// SIMATIC S7-200 project (STEP 7-Micro/WIN), CPU 216 REL 01.02

SYMBOL_TABLE USR1
Always_On        SM0.0    // This bit is always on.
First_Scan_On    SM0.1    // This bit is on for the first scan cycle only.
Clock_1s         SM0.5    // Clock pulse that is on for 0.5 s, off for 0.5 s, for a duty cycle time of 1 s.
Down_Bit         M0.0     // This "count down" memory bit determines the counting direction.
END_SYMBOL_TABLE

ORGANIZATION_BLOCK MAIN:OB1
TITLE= Tip002B
//  题目： 处理输入/输出中断
// ***概述***
// 本程序适用于SIMATIC S7-212和S7-214的计数器，可以从0计到255，这要取决于输入I0.0
// 的状态。如果将输入I0.0置为1，则程序减计数；如果将输入I0.0置为0，则程序加计数
// 如果输入I0.0的状态改变，则将立即激活输入/输出中断程序，中断程序0或1分别将存储器位M0.0
// 置成1或0。
// ***程序和注释***
// 本程序是一个输入/输出中断程序的范例，计数器从0计到255。如果输入I0.0
// 为0，则程序加计数，如果输入I0.0为1，则程序减计数。
// 本程序包括以下三个程序：
// Main  （主程序）            初始化和计数
// INT0   （中断程序0）        输入I0.0为1时，减计数。
// INT1   （中断程序1）        输入I0.0为0时，加计数。
// 本程序长度为32个字。
// 标题：事件中断
// 
BEGIN
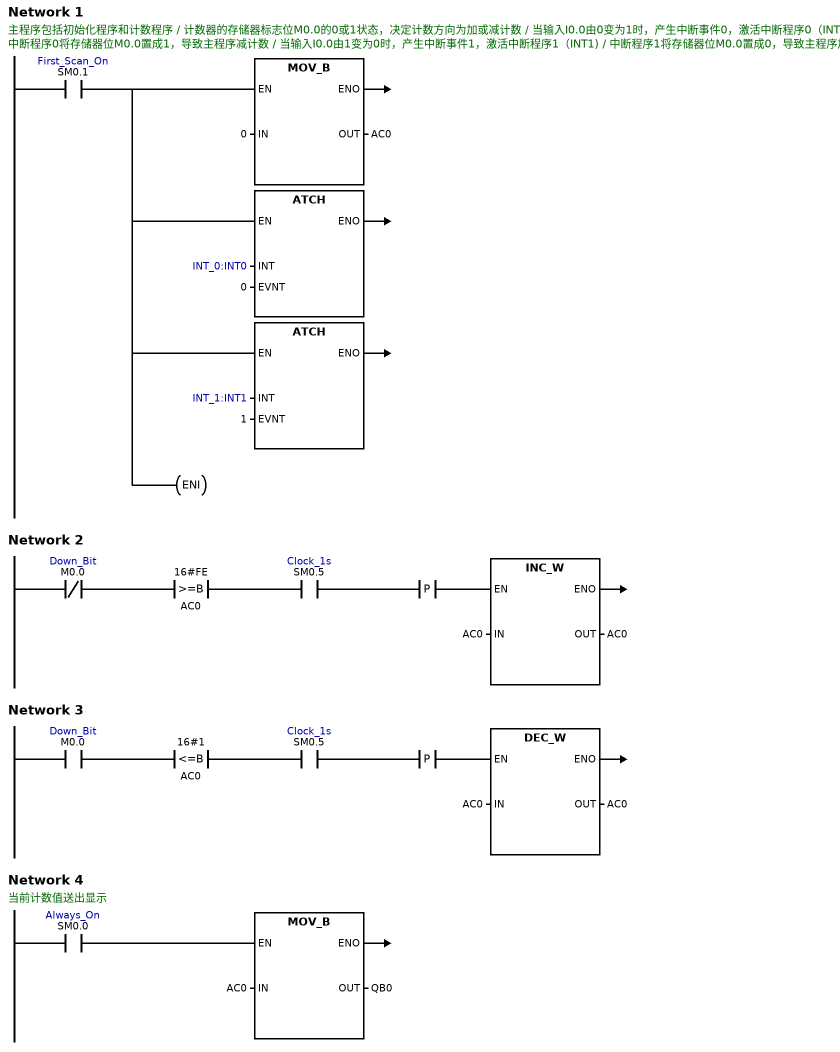
Network 1
// 主程序包括初始化程序和计数程序
// 计数器的存储器标志位M0.0的0或1状态，决定计数方向为加或减计数
// 当输入I0.0由0变为1时，产生中断事件0，激活中断程序0（INT0）
// 中断程序0将存储器位M0.0置成1，导致主程序减计数
// 当输入I0.0由1变为0时，产生中断事件1，激活中断程序1（INT1)
// 中断程序1将存储器位M0.0置成0，导致主程序加计数
// 仅首次扫描时，SM0.1才为1，进行以下初始化
//将计数累加器AC0清0
//输入I0.0为上升沿时激活事件中断0
//输入I0.0为上升沿时激活事件中断1
//允许中断
LD     First_Scan_On:SM0.1
MOVB   0, AC0
ATCH   INT_0:INT0, 0
ATCH   INT_1:INT1, 1
ENI
Network 2
//如果存储器的标志位M0.0为0状态
//且计数累加器AC0的当前计数值小于或等于254
//且0.5秒脉冲
// 且上升沿
//那么计数累加器AC0加1
// (network saved uncompiled; LAD cells follow)
// row 0: c0 -|/|- Down_Bit:M0.0  c1 -|>=B|- 16#FE, AC0  c2 -| |- Clock_1s:SM0.5  c3 -|P|-  c4 [INC_W EN:=power@row0, IN:=AC0, ENO=>power, OUT=>AC0]  c5 ->
// row 1: c4 [box]
Network 3
// 如果存储器的标志位M0.0为1状态 
// 且计数累加器AC0的当前计数值大于或等于1
// 且0.5秒脉冲
// 且上升沿
//那么计数累加器AC0减1
// (network saved uncompiled; LAD cells follow)
// row 0: c0 -| |- Down_Bit:M0.0  c1 -|<=B|- 16#1, AC0  c2 -| |- Clock_1s:SM0.5  c3 -|P|-  c4 [DEC_W EN:=power@row0, IN:=AC0, ENO=>power, OUT=>AC0]  c5 ->
// row 1: c4 [box]
Network 4
// 当前计数值送出显示
// SM0.0总是1
//在输出端Q0.0至Q0.7显示AC0的当前计数值
LD     Always_On:SM0.0
MOVB   AC0, QB0
Network 5 // 主程序结束
// MEND
// 
Network 6 // ***中断程序0 ***
// 事件中断程序0将存储器的标志位M0.0置成1
// 此情况下程序减计数
// 
END_ORGANIZATION_BLOCK

INTERRUPT_BLOCK INT_0:INT0
TITLE=
BEGIN
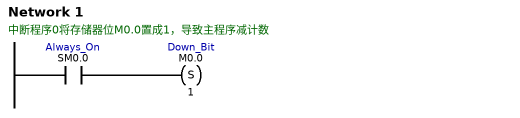
Network 1
// 中断程序0将存储器位M0.0置成1，导致主程序减计数
// SM0.0总是1
// 将存储器的标志位M0.0置成1
LD     Always_On:SM0.0
S      Down_Bit:M0.0, 1
Network 2 //  中断程序0结束
// RETI
// 
END_INTERRUPT_BLOCK

INTERRUPT_BLOCK INT_1:INT1
TITLE=
BEGIN
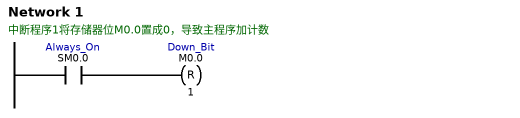
Network 1
// 中断程序1将存储器位M0.0置成0，导致主程序加计数
// SM0.0总是1.
// 将存储器的标志位M0.0置成0
LD     Always_On:SM0.0
R      Down_Bit:M0.0, 1
Network 2 // 中断程序1结束
// RETI
// 
END_INTERRUPT_BLOCK
